(* PLC project SansNom, Inconnu SansNom 1 *)
(* stored: creationDateTime 2023-11-29T19:20:17, modificationDateTime 2023-11-29T19:45:09 *)

(* CONTROL *)
PROGRAM program0
  VAR
    RED : BOOL;
    YELLOW : BOOL;
    GREEN : BOOL;
    CONTROL : BOOL;
    INPUT : BOOL;
    TP0 : TP;
    TP1 : TP;
    TP2 : TP;
    TP3 : TP;
  END_VAR

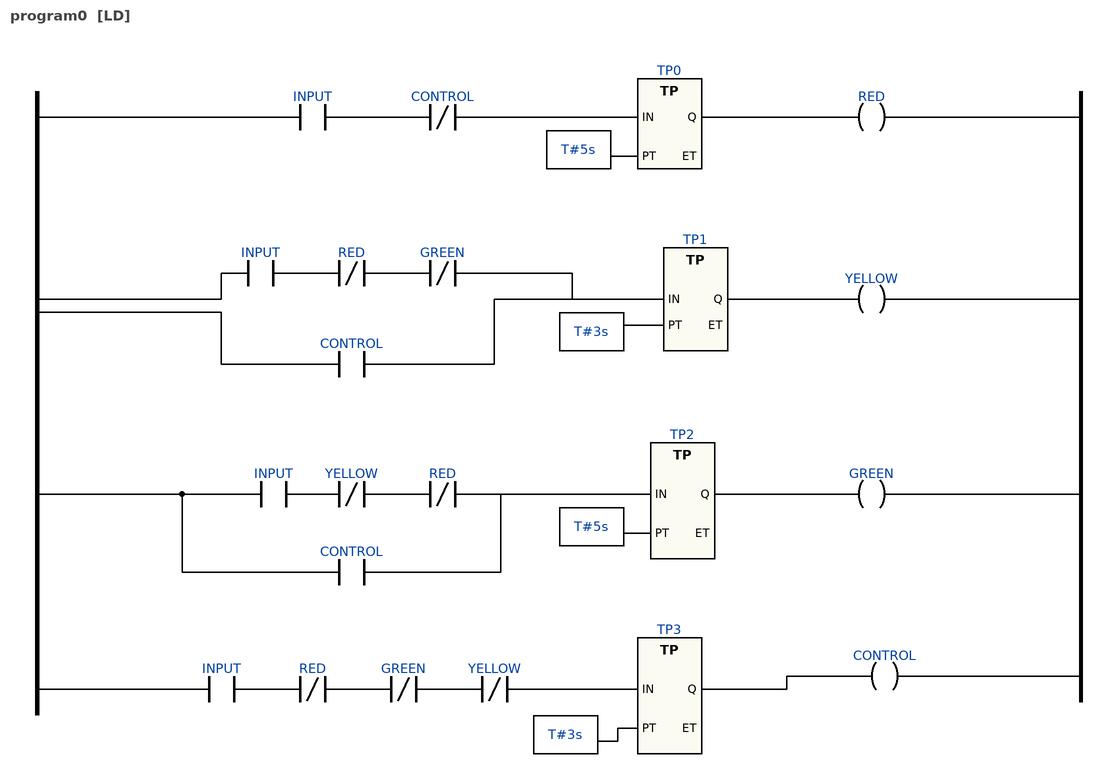
(* LD diagram, written out as Structured Text *)
TP0(IN := INPUT AND NOT CONTROL, PT := T#5s);
RED := TP0.Q;
TP1(IN := CONTROL OR INPUT AND NOT RED AND NOT GREEN, PT := T#3s);
YELLOW := TP1.Q;
TP2(IN := CONTROL OR INPUT AND NOT YELLOW AND NOT RED, PT := T#5s);
GREEN := TP2.Q;
TP3(IN := INPUT AND NOT RED AND NOT GREEN AND NOT YELLOW, PT := T#3s);
CONTROL := TP3.Q;
END_PROGRAM

CONFIGURATION Config0
  RESOURCE Res0 ON PLC
    TASK task0(INTERVAL := T#20ms, PRIORITY := 0);
    PROGRAM instance0 WITH task0 : program0;
  END_RESOURCE
END_CONFIGURATION
